// TIA Portal V15.1 export
// export: Created 2020-06-12T07:35:49.3193359Z, ExportSetting None, DisplayName Totally Integrated Automation Portal, DisplayVersion V15.1, DisplayName TIA Portal Openness, DisplayVersion V15.1, DisplayName STEP 7 Professional, DisplayVersion V15.1, DisplayName STEP 7 Safety, DisplayVersion V15.1, DisplayName WinCC Advanced, DisplayVersion V15.1
FUNCTION "HOOD_seal" : Void   // FC109, FBD
TITLE = Hood Sealing
{ S7_Optimized_Access := 'FALSE' }
// stored: SetENOAutomatically False
   VAR_TEMP
      _no_pos : Bool;
      _csf : Bool;
      tSealEna : Bool;
      tQ1 : Bool;
      tQ2 : Bool;
      tQ3 : Bool;
      tBypass : Bool;
      tBool : Bool;
      tSubReq : Bool;
      tHmiSealOn : Bool;
      tHmiSealOff : Bool;
      tSealIsOn : Bool;
      tSealIsOff : Bool;
   END_VAR
BEGIN

REGION Network 1: Common System Fault
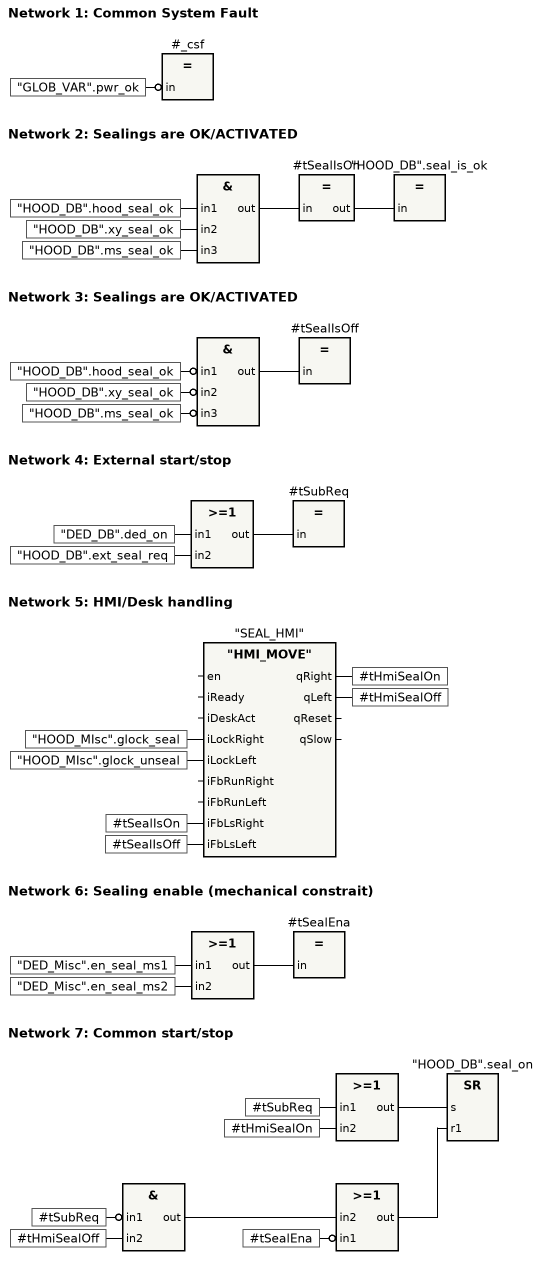
   #_csf := NOT "GLOB_VAR".pwr_ok;
END_REGION

REGION Network 2: Sealings are OK/ACTIVATED
   #tSealIsOn := "HOOD_DB".hood_seal_ok AND "HOOD_DB".xy_seal_ok AND "HOOD_DB".ms_seal_ok;
   "HOOD_DB".seal_is_ok := #tSealIsOn;
END_REGION

REGION Network 3: Sealings are OK/ACTIVATED
   #tSealIsOff := NOT "HOOD_DB".hood_seal_ok AND NOT "HOOD_DB".xy_seal_ok AND NOT "HOOD_DB".ms_seal_ok;
END_REGION

REGION Network 4: External start/stop
   #tSubReq := "DED_DB".ded_on OR "HOOD_DB".ext_seal_req;
END_REGION

REGION Network 5: HMI/Desk handling
   "SEAL_HMI"(iLockRight := "HOOD_MIsc".glock_seal,   // "HMI_MOVE"
              iLockLeft := "HOOD_MIsc".glock_unseal,
              iFbLsRight := #tSealIsOn,
              iFbLsLeft := #tSealIsOff,
              qRight => #tHmiSealOn,
              qLeft => #tHmiSealOff);
END_REGION

REGION Network 6: Sealing enable (mechanical constrait)
   #tSealEna := "DED_Misc".en_seal_ms1 OR "DED_Misc".en_seal_ms2;
END_REGION

REGION Network 7: Common start/stop
   IF #tSubReq OR #tHmiSealOn THEN
       "HOOD_DB".seal_on := TRUE;   // SR flip-flop
   END_IF;
   IF (NOT #tSubReq AND #tHmiSealOff) OR NOT #tSealEna THEN "HOOD_DB".seal_on := FALSE; END_IF;
END_REGION

REGION Network 8: MS1: Enable sealing
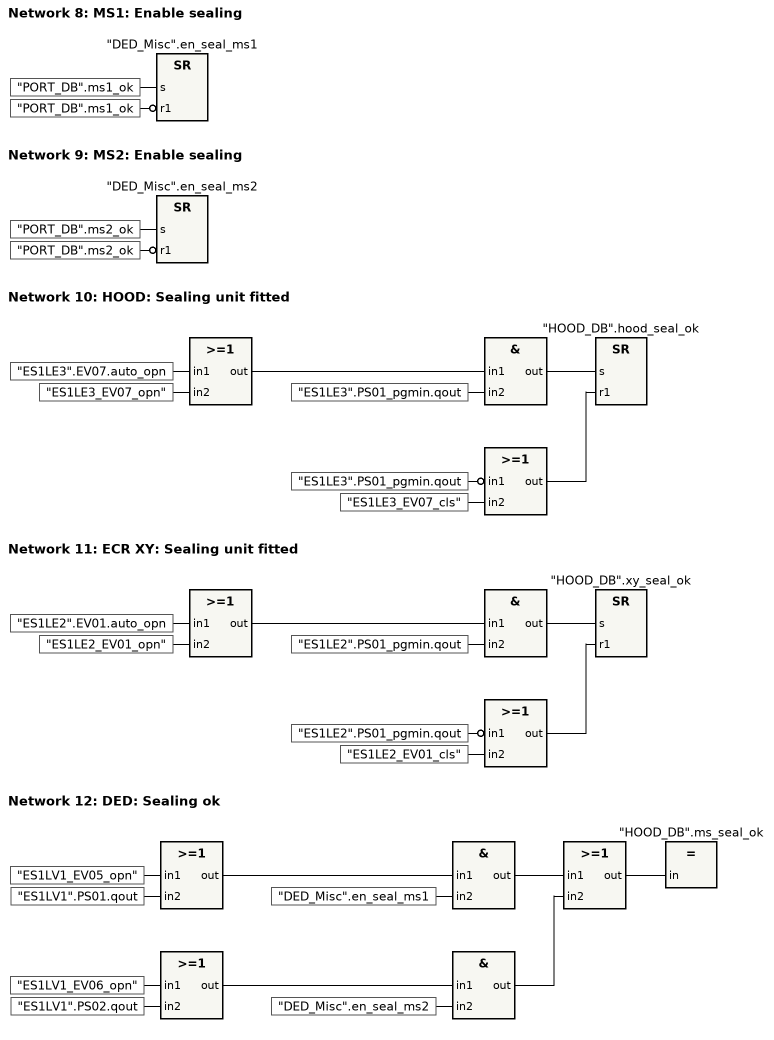
   IF "PORT_DB".ms1_ok THEN
       "DED_Misc".en_seal_ms1 := TRUE;   // SR flip-flop
   END_IF;
   IF NOT "PORT_DB".ms1_ok THEN "DED_Misc".en_seal_ms1 := FALSE; END_IF;
END_REGION

REGION Network 9: MS2: Enable sealing
   IF "PORT_DB".ms2_ok THEN
       "DED_Misc".en_seal_ms2 := TRUE;   // SR flip-flop
   END_IF;
   IF NOT "PORT_DB".ms2_ok THEN "DED_Misc".en_seal_ms2 := FALSE; END_IF;
END_REGION

REGION Network 10: HOOD: Sealing unit fitted
   IF ("ES1LE3".EV07.auto_opn OR "ES1LE3_EV07_opn") AND "ES1LE3".PS01_pgmin.qout THEN
       "HOOD_DB".hood_seal_ok := TRUE;   // SR flip-flop
   END_IF;
   IF NOT "ES1LE3".PS01_pgmin.qout OR "ES1LE3_EV07_cls" THEN "HOOD_DB".hood_seal_ok := FALSE; END_IF;
END_REGION

REGION Network 11: ECR XY: Sealing unit fitted
   IF ("ES1LE2".EV01.auto_opn OR "ES1LE2_EV01_opn") AND "ES1LE2".PS01_pgmin.qout THEN
       "HOOD_DB".xy_seal_ok := TRUE;   // SR flip-flop
   END_IF;
   IF NOT "ES1LE2".PS01_pgmin.qout OR "ES1LE2_EV01_cls" THEN "HOOD_DB".xy_seal_ok := FALSE; END_IF;
END_REGION

REGION Network 12: DED: Sealing ok
   "HOOD_DB".ms_seal_ok := (("ES1LV1_EV05_opn" OR "ES1LV1".PS01.qout) AND "DED_Misc".en_seal_ms1) OR (("ES1LV1_EV06_opn" OR "ES1LV1".PS02.qout) AND "DED_Misc".en_seal_ms2);
END_REGION

REGION Network 13: Sealing LOCK (close/activate)
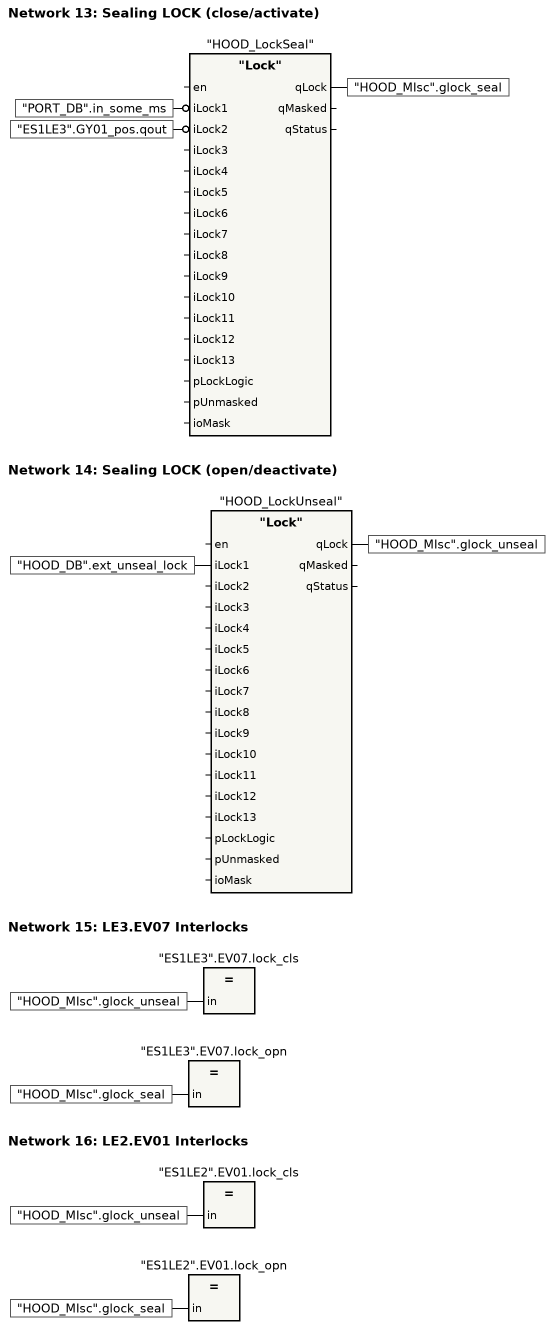
   "HOOD_LockSeal"(iLock1 := NOT "PORT_DB".in_some_ms,   // "Lock"
                   iLock2 := NOT "ES1LE3".GY01_pos.qout,
                   qLock => "HOOD_MIsc".glock_seal);
END_REGION

REGION Network 14: Sealing LOCK (open/deactivate)
   "HOOD_LockUnseal"(iLock1 := "HOOD_DB".ext_unseal_lock, qLock => "HOOD_MIsc".glock_unseal);   // "Lock"
END_REGION

REGION Network 15: LE3.EV07 Interlocks
   "ES1LE3".EV07.lock_cls := "HOOD_MIsc".glock_unseal;
   "ES1LE3".EV07.lock_opn := "HOOD_MIsc".glock_seal;
END_REGION

REGION Network 16: LE2.EV01 Interlocks
   "ES1LE2".EV01.lock_cls := "HOOD_MIsc".glock_unseal;
   "ES1LE2".EV01.lock_opn := "HOOD_MIsc".glock_seal;
END_REGION

REGION Network 17: ES1LV1.EV05, MS1 sealing: Interlocks
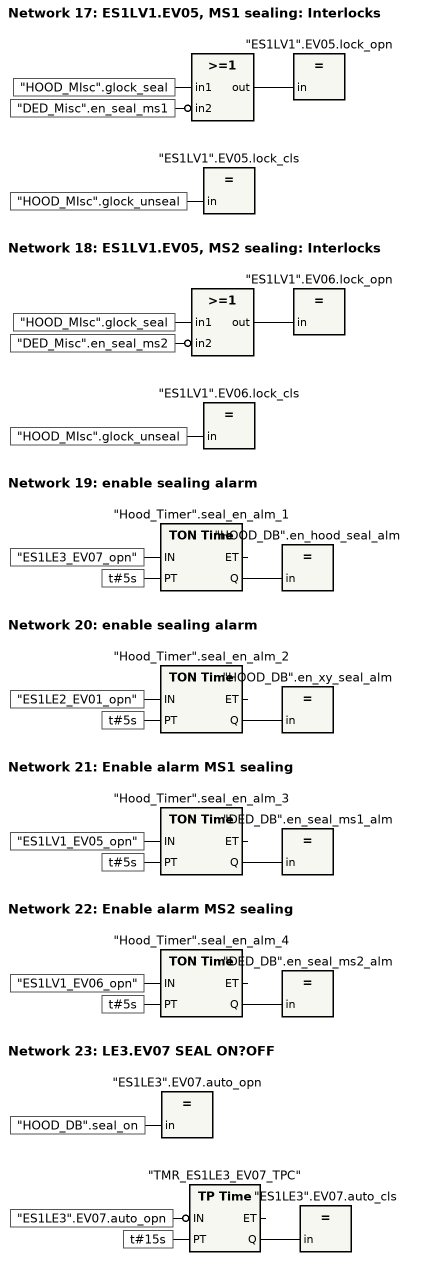
   "ES1LV1".EV05.lock_opn := "HOOD_MIsc".glock_seal OR NOT "DED_Misc".en_seal_ms1;
   "ES1LV1".EV05.lock_cls := "HOOD_MIsc".glock_unseal;
END_REGION

REGION Network 18: ES1LV1.EV05, MS2 sealing: Interlocks
   "ES1LV1".EV06.lock_opn := "HOOD_MIsc".glock_seal OR NOT "DED_Misc".en_seal_ms2;
   "ES1LV1".EV06.lock_cls := "HOOD_MIsc".glock_unseal;
END_REGION

REGION Network 19: enable sealing alarm
   "Hood_Timer".seal_en_alm_1.TON(IN := "ES1LE3_EV07_opn", PT := t#5s);
   "HOOD_DB".en_hood_seal_alm := "Hood_Timer".seal_en_alm_1.Q;
END_REGION

REGION Network 20: enable sealing alarm
   "Hood_Timer".seal_en_alm_2.TON(IN := "ES1LE2_EV01_opn", PT := t#5s);
   "HOOD_DB".en_xy_seal_alm := "Hood_Timer".seal_en_alm_2.Q;
END_REGION

REGION Network 21: Enable alarm MS1 sealing
   "Hood_Timer".seal_en_alm_3.TON(IN := "ES1LV1_EV05_opn", PT := t#5s);
   "DED_DB".en_seal_ms1_alm := "Hood_Timer".seal_en_alm_3.Q;
END_REGION

REGION Network 22: Enable alarm MS2 sealing
   "Hood_Timer".seal_en_alm_4.TON(IN := "ES1LV1_EV06_opn", PT := t#5s);
   "DED_DB".en_seal_ms2_alm := "Hood_Timer".seal_en_alm_4.Q;
END_REGION

REGION Network 23: LE3.EV07 SEAL ON?OFF
   "ES1LE3".EV07.auto_opn := "HOOD_DB".seal_on;
   "TMR_ES1LE3_EV07_TPC".TP(IN := NOT "ES1LE3".EV07.auto_opn, PT := t#15s);
   "ES1LE3".EV07.auto_cls := "TMR_ES1LE3_EV07_TPC".Q;
END_REGION

REGION Network 24: LE2.EV01 SEAL ON?OFF
   // ES1LE3_EV07.auto_opn
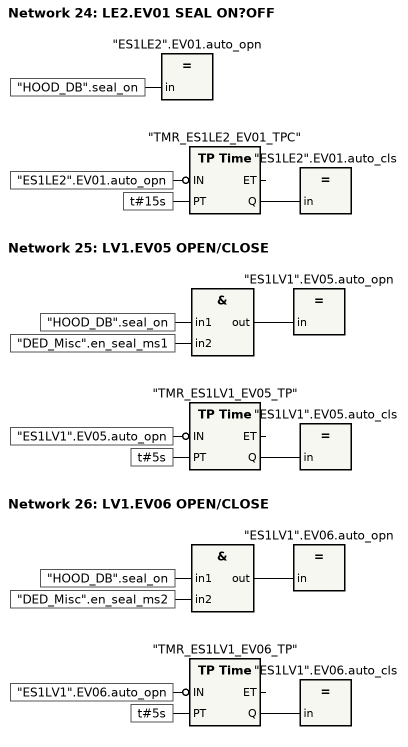
   "ES1LE2".EV01.auto_opn := "HOOD_DB".seal_on;
   "TMR_ES1LE2_EV01_TPC".TP(IN := NOT "ES1LE2".EV01.auto_opn, PT := t#15s);
   "ES1LE2".EV01.auto_cls := "TMR_ES1LE2_EV01_TPC".Q;
END_REGION

REGION Network 25: LV1.EV05 OPEN/CLOSE
   "ES1LV1".EV05.auto_opn := "HOOD_DB".seal_on AND "DED_Misc".en_seal_ms1;
   "TMR_ES1LV1_EV05_TP".TP(IN := NOT "ES1LV1".EV05.auto_opn, PT := t#5s);
   "ES1LV1".EV05.auto_cls := "TMR_ES1LV1_EV05_TP".Q;
END_REGION

REGION Network 26: LV1.EV06 OPEN/CLOSE
   "ES1LV1".EV06.auto_opn := "HOOD_DB".seal_on AND "DED_Misc".en_seal_ms2;
   "TMR_ES1LV1_EV06_TP".TP(IN := NOT "ES1LV1".EV06.auto_opn, PT := t#5s);
   "ES1LV1".EV06.auto_cls := "TMR_ES1LV1_EV06_TP".Q;
END_REGION

REGION Network 27: [[end]]
END_REGION
END_FUNCTION
